PROGRAM Tools
VAR
END_VAR

METHOD inToleranz : BOOL
VAR_INPUT
	fIstwert:		REAL;
	fMin:			REAL;
	fMax:			REAL;
END_VAR
inToleranz := fIstwert >= fMin AND fIstwert <= fMax;
END_METHOD

METHOD runden : REAL
VAR_INPUT
	fInput:			REAL;
	nAnzStellen:	DINT;
END_VAR

VAR
	nZwResultat:	DINT;
END_VAR
nZwResultat := REAL_TO_DINT(fInput*EXPT(10,nAnzStellen+1));
IF 			(nZwResultat MOD 10) >= 5THEN
	nZwResultat := nZwResultat + 10;
END_IF
nZwResultat := nZwResultat / 10;
runden		:= DINT_TO_REAL(nZwResultat)/EXPT(10,nAnzStellen);
END_METHOD

END_PROGRAM

(* stored: Version 1.1.0.1, ProductVersion 3.1.4024.12
   POU Tools: Id {30ed2c2e-5277-45ca-b09f-479539575525}, SpecialFunc None
   Method inToleranz: Id {5d2bf1ed-903e-4a2c-abac-faade7c10ba8}
   Method runden: Id {d083471d-cb39-46e1-9e8f-d8cbf287e138} *)
